PROGRAM MAIN

ALIAS();
ANALOGconversion();
handleFAULT();
handlesensorlimitFAULTS();
handlesoftEXCEPTION();
Automated_Capacitor_Test_ST();	
HMI();
HV_Monitor();
VoltMonitor();
// runningLIGHTS();

END_PROGRAM

(* stored: Version 1.1.0.1, ProductVersion 3.1.4024.11
   POU MAIN: Id {c44dd456-9fdd-4969-ac7e-7e1422e6d84f}, SpecialFunc None *)
